// TIA Portal V19 export
DATA_BLOCK "Config"   // DB166
// stored: MemoryReserve 100, Namespace Unit.Em2
   VAR
      em { ExternalWritable := 'False'} : "LAF_typeEmConfiguration";   // Configuration of EM Parameters
      axis { ExternalWritable := 'False'} : Array[1.._.EM2_NO_OF_AXES] of DB_ANY;   // Assign the axis of the EM
   END_VAR
BEGIN
   em.referenceDesignator.parent := WSTRING#'Unit';
   em.referenceDesignator.relative := WSTRING#'EM2 HighPerfMotion';
END_DATA_BLOCK
